// TIA Portal V18 export
FUNCTION_BLOCK "Multi instance FB"   // FB2, LAD
{ S7_Optimized_Access := 'TRUE' }
VERSION : 0.1
// stored: AutoNumber true, IsIECCheckEnabled false, IsRetainMemResEnabled false, MemoryReserve 100, SetENOAutomatically false, UDAEnableTagReadback false
   VAR
      "Motor control function FB_Instance" { S7_SetPoint := 'True'} : "Motor control function FB";
      "Motor control function FB_Instance_1" { S7_SetPoint := 'True'} : "Motor control function FB";
   END_VAR
BEGIN

REGION Network 1: Motor 1
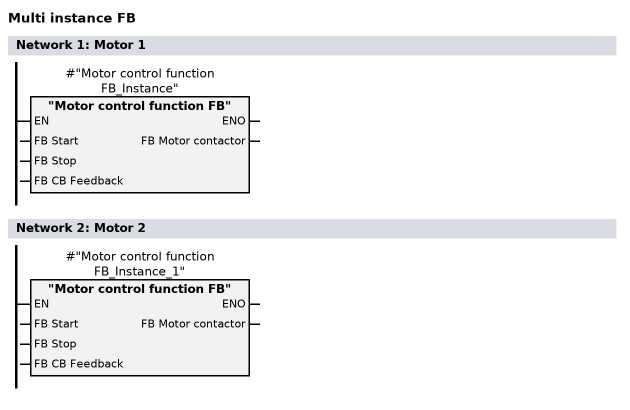
   RUNG wire#powerrail
      #"Motor control function FB_Instance"("FB Start" :=, "FB Stop" :=, "FB CB Feedback" :=, "FB Motor contactor" =>)
   END_RUNG
   // the same network as SCL:
   #"Motor control function FB_Instance"();   // "Motor control function FB"
END_REGION

REGION Network 2: Motor 2
   RUNG wire#powerrail
      #"Motor control function FB_Instance_1"("FB Start" :=, "FB Stop" :=, "FB CB Feedback" :=, "FB Motor contactor" =>)
   END_RUNG
   // the same network as SCL:
   #"Motor control function FB_Instance_1"();   // "Motor control function FB"
END_REGION
END_FUNCTION_BLOCK
